(* Schneider Machine Expert - Basic project MKH simpang 5, file version 1.7.0.0 *)
(* ProjectInformations: Name=New project *)

HARDWARE
  Cpu 0: TM221ME32TK
  EthernetConfiguration: NetworkName=M221, IpAllocationMode=FixedAddress, IpAddress=0.0.0.0, SubnetMask=0.0.0.0
  SerialLineConfiguration: Baud=Baud19200, Parity=ParityEven, DataBits=DataBits8, StopBits=StopBits1, PhysicalMedium=PhysicalMediumRs485, TransmissionMode=TransmissionModeModbusRtu, SlaveId=1, Addressing=SlaveAddressing
  MastTask: UsePeriodScanMode=false, PeriodScan=100
  FastTask: Period=255
  CpuBehavior: StartingMode=StartAsPreviousState, AutoSaveRamOnEeprom=true, WatchdogPeriod=250

SYMBOLS  (address, symbol, comment, settings)
  %M1         "M1"
  %TM1        "T1"  [Preset=3, Base=OneSecond]
  %TM2        "T2"  [Preset=1, Base=OneSecond]
  %TM3        "T3"  [Preset=3, Base=OneSecond]
  %TM4        "T4"  [Preset=1, Base=OneSecond]
  %TM5        "T5"  [Preset=3, Base=OneSecond]
  %TM6        "T6"  [Preset=1, Base=OneSecond]
  %TM7        "T7"  [Preset=3, Base=OneSecond]
  %TM8        "T8"  [Preset=1, Base=OneSecond]
  %TM9        "T9"  [Preset=3, Base=OneSecond]
  %TM10       "T10"  [Preset=1, Base=OneSecond]
  %I0.0       "S1"
  %Q0.1       "Hi 1"
  %Q0.2       "Ku 1"
  %Q0.3       "Me 1"
  %Q0.4       "Hi 2"
  %Q0.5       "Ku 2"
  %Q0.6       "Me 2"
  %Q0.7       "Hi 3"
  %Q0.8       "Ku 3"
  %Q0.9       "Me 3"
  %Q0.10      "Hi 4"
  %Q0.11      "Ku 4"
  %Q0.12      "Me 4"
  %Q0.13      "Hi 5"
  %Q0.14      "Ku 5"
  %Q0.15      "Me 5"

POU New POU
  (* SectionNumber=1 *)

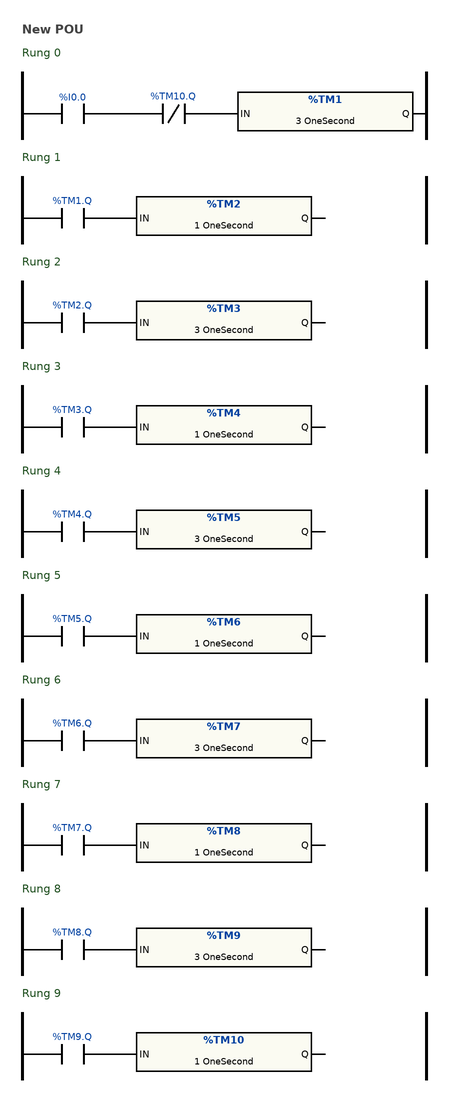

// Rung 0
  BLK %TM1
  LD %I0.0
  ANDN %TM10.Q
  IN
  END_BLK
  // as ST:
  //   %TM1(IN := %I0.0 AND NOT %TM10.Q);

// Rung 1
  BLK %TM2
  LD %TM1.Q
  IN
  END_BLK
  // as ST:
  //   %TM2(IN := %TM1.Q);

// Rung 2
  BLK %TM3
  LD %TM2.Q
  IN
  END_BLK
  // as ST:
  //   %TM3(IN := %TM2.Q);

// Rung 3
  BLK %TM4
  LD %TM3.Q
  IN
  END_BLK
  // as ST:
  //   %TM4(IN := %TM3.Q);

// Rung 4
  BLK %TM5
  LD %TM4.Q
  IN
  END_BLK
  // as ST:
  //   %TM5(IN := %TM4.Q);

// Rung 5
  BLK %TM6
  LD %TM5.Q
  IN
  END_BLK
  // as ST:
  //   %TM6(IN := %TM5.Q);

// Rung 6
  BLK %TM7
  LD %TM6.Q
  IN
  END_BLK
  // as ST:
  //   %TM7(IN := %TM6.Q);

// Rung 7
  BLK %TM8
  LD %TM7.Q
  IN
  END_BLK
  // as ST:
  //   %TM8(IN := %TM7.Q);

// Rung 8
  BLK %TM9
  LD %TM8.Q
  IN
  END_BLK
  // as ST:
  //   %TM9(IN := %TM8.Q);

// Rung 9
  BLK %TM10
  LD %TM9.Q
  IN
  END_BLK
  // as ST:
  //   %TM10(IN := %TM9.Q);

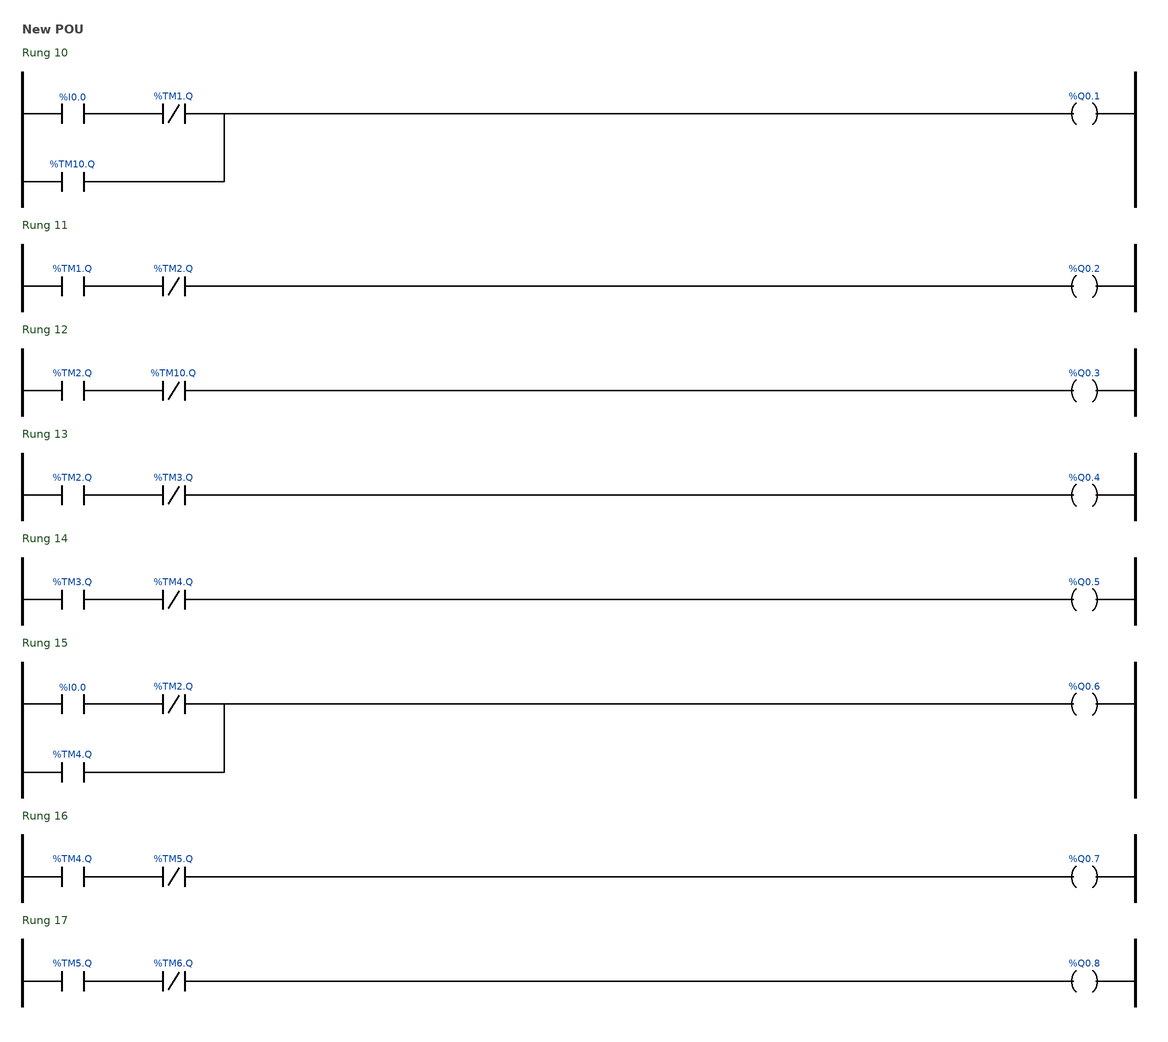

// Rung 10
  LD %I0.0
  ANDN %TM1.Q
  OR %TM10.Q
  ST %Q0.1
  // as ST:
  //   %Q0.1 := %I0.0 AND NOT %TM1.Q OR %TM10.Q;

// Rung 11
  LD %TM1.Q
  ANDN %TM2.Q
  ST %Q0.2
  // as ST:
  //   %Q0.2 := %TM1.Q AND NOT %TM2.Q;

// Rung 12
  LD %TM2.Q
  ANDN %TM10.Q
  ST %Q0.3
  // as ST:
  //   %Q0.3 := %TM2.Q AND NOT %TM10.Q;

// Rung 13
  LD %TM2.Q
  ANDN %TM3.Q
  ST %Q0.4
  // as ST:
  //   %Q0.4 := %TM2.Q AND NOT %TM3.Q;

// Rung 14
  LD %TM3.Q
  ANDN %TM4.Q
  ST %Q0.5
  // as ST:
  //   %Q0.5 := %TM3.Q AND NOT %TM4.Q;

// Rung 15
  LD %I0.0
  ANDN %TM2.Q
  OR %TM4.Q
  ST %Q0.6
  // as ST:
  //   %Q0.6 := %I0.0 AND NOT %TM2.Q OR %TM4.Q;

// Rung 16
  LD %TM4.Q
  ANDN %TM5.Q
  ST %Q0.7
  // as ST:
  //   %Q0.7 := %TM4.Q AND NOT %TM5.Q;

// Rung 17
  LD %TM5.Q
  ANDN %TM6.Q
  ST %Q0.8
  // as ST:
  //   %Q0.8 := %TM5.Q AND NOT %TM6.Q;

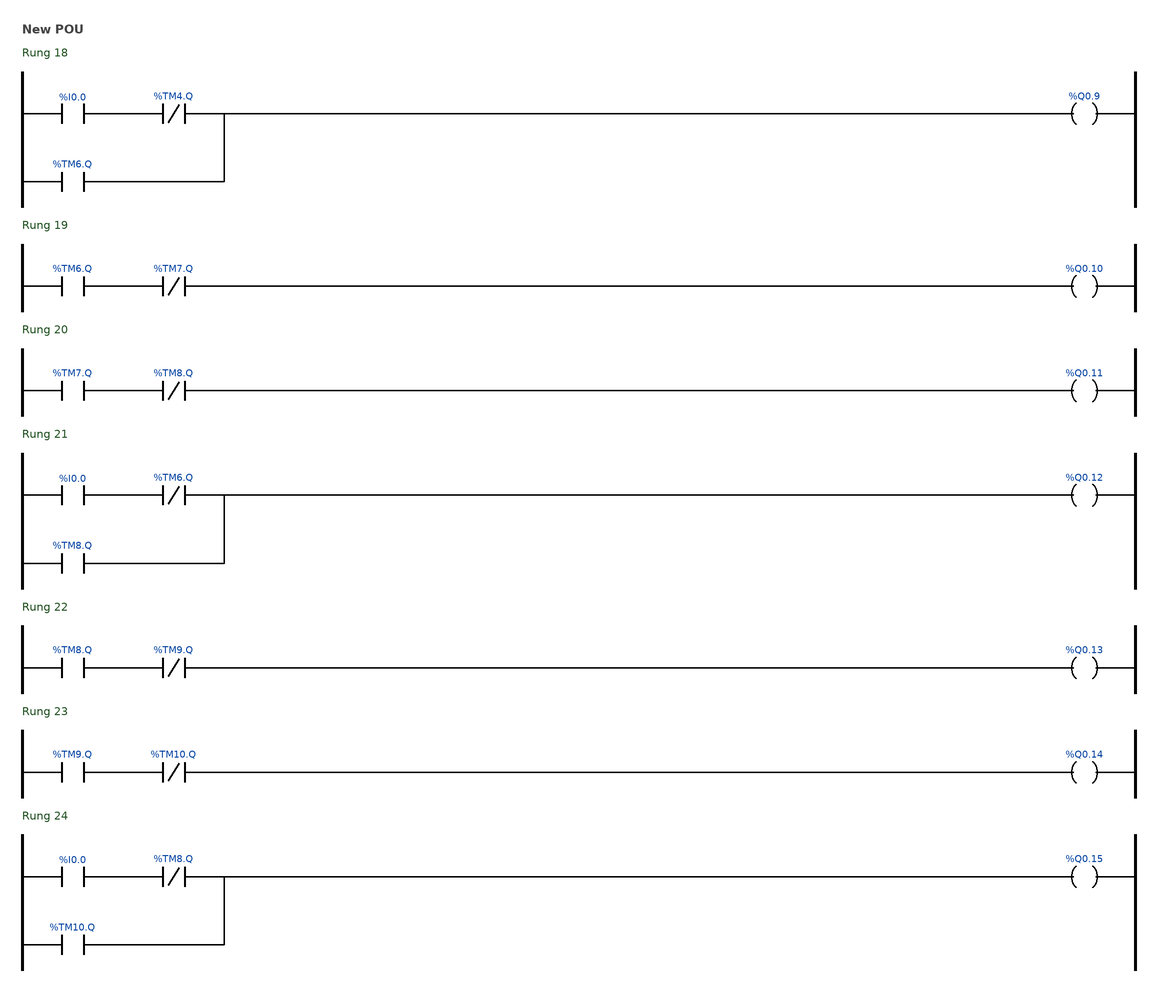

// Rung 18
  LD %I0.0
  ANDN %TM4.Q
  OR %TM6.Q
  ST %Q0.9
  // as ST:
  //   %Q0.9 := %I0.0 AND NOT %TM4.Q OR %TM6.Q;

// Rung 19
  LD %TM6.Q
  ANDN %TM7.Q
  ST %Q0.10
  // as ST:
  //   %Q0.10 := %TM6.Q AND NOT %TM7.Q;

// Rung 20
  LD %TM7.Q
  ANDN %TM8.Q
  ST %Q0.11
  // as ST:
  //   %Q0.11 := %TM7.Q AND NOT %TM8.Q;

// Rung 21
  LD %I0.0
  ANDN %TM6.Q
  OR %TM8.Q
  ST %Q0.12
  // as ST:
  //   %Q0.12 := %I0.0 AND NOT %TM6.Q OR %TM8.Q;

// Rung 22
  LD %TM8.Q
  ANDN %TM9.Q
  ST %Q0.13
  // as ST:
  //   %Q0.13 := %TM8.Q AND NOT %TM9.Q;

// Rung 23
  LD %TM9.Q
  ANDN %TM10.Q
  ST %Q0.14
  // as ST:
  //   %Q0.14 := %TM9.Q AND NOT %TM10.Q;

// Rung 24
  LD %I0.0
  ANDN %TM8.Q
  OR %TM10.Q
  ST %Q0.15
  // as ST:
  //   %Q0.15 := %I0.0 AND NOT %TM8.Q OR %TM10.Q;
